PROGRAM MAIN
VAR
	nAlive: INT;
	breset: BOOL;
	nDemoVariable : INT;
	nCX8200_State	AT %I*	: UINT;
END_VAR

VAR PERSISTENT
	nDemoVar_Persist: INT;
END_VAR

nAlive:= nAlive + 1;
GVL_AHDataModbus.nCX8200_State_MB := nCX8200_State;

//Håndterer vedvarende data
	P_SystemDK.M_nCyclic(bReset := breset );
//Håndterer DALI-diagnostik (run once)
	P_DALI_DIAG();
//Håndterer adressering		
	DALI_Commissioning();
//Håndterer energirapportering
	P_DALI_Energy_Line();
//Håndterer moodbus-kommunikation (kun PLC-oversigt)
	P_AHModbusComm();

//Håndterer individuel lyskontrol i lokaler
	//Gange
	P_Gang_3_409();
	P_Gang_4_410A();
	P_Gang_4_413();

	
	//Rum
	P_Rum_3_429();
	P_Rum_4_407();
	P_Rum_4_411();
	
//Testprogrammer
	//P_DALI_Energy_Firmware_Test();

END_PROGRAM

(* stored: Version 1.1.0.1
   POU MAIN: Id {6bf17237-b1a6-4c57-bf47-1238f1ca1a56}, SpecialFunc None *)
